Omron CX-Programmer project NewProject (CX-Programmer 9.75)

# PLC NewPLC1: CP1L M

## Global symbols (name address type ; comment)
0.00 BOOL  ; PB ON 1
0.01 BOOL  ; PB OFF 1
0.02 BOOL  ; PB ON 2
0.03 BOOL  ; PB OFF 2
0.04 BOOL  ; PB ON 3
0.05 BOOL  ; PB OFF 3
100.00 BOOL  ; K1
100.01 BOOL  ; K2
100.02 BOOL  ; K3

## Program NewProgram1 (cyclic task 0)
Local symbols
tm3 UINT

### Section Berurutan

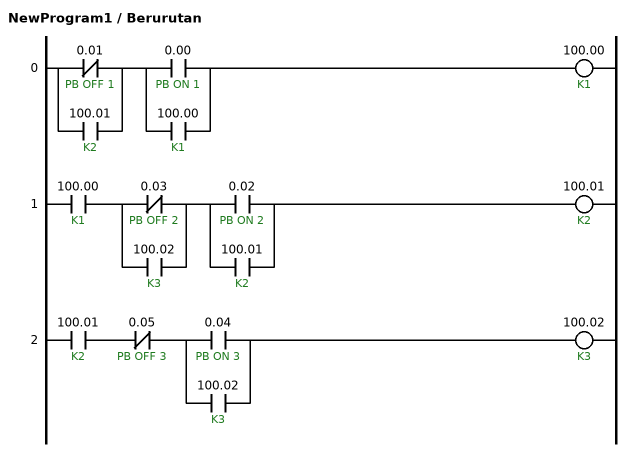
; rung 0
LDNOT 0.01  ; PB OFF 1
OR 100.01  ; K2
LD 0.00  ; PB ON 1
OR 100.00  ; K1
ANDLD
OUT 100.00  ; K1
; rung 1
LD 100.00  ; K1
LDNOT 0.03  ; PB OFF 2
OR 100.02  ; K3
ANDLD
LD 0.02  ; PB ON 2
OR 100.01  ; K2
ANDLD
OUT 100.01  ; K2
; rung 2
LD 100.01  ; K2
ANDNOT 0.05  ; PB OFF 3
LD 0.04  ; PB ON 3
OR 100.02  ; K3
ANDLD
OUT 100.02  ; K3

### Section END
; rung 0
END(001)